KUKA KRL program: TRIGBACK.src

&ACCESS RV
&REL 3
&PARAM TEMPLATE = C:\KRC\Roboter\Template\FunctionVorgabe
&PARAM EDITMASK = *
DEFFCT BOOL TRIGBACK( )

DECL STIFFNESS USERSTIFF

DECL INT md_int[16]
DECL REAL md_real[16]
DECL INT n
DECL INT result

;USERSTIFF=$STIFFNESS
;USERSTIFF.STRATEGY=10
;USERSTIFF.FRAMETYPE=#TOOL
;USERSTIFF.TOOL={X 0.0,Y 0.0,Z 180.0,A 0.0,B 0.0,C 0.0}
;USERSTIFF.CPSTIFFNESS={X 2000,Y 2000,Z 2000,A 200,B 200,C 200}
;USERSTIFF.CPDAMPING={X 0.7,Y 0.7,Z 0.7,A 0.7,B 0.7,C 0.7}
;USERSTIFF.AXISSTIFFNESS={A1 2000,A2 2000,A3 2000,A4 2000,A5 2000,A6 2000,E1 2000}
;USERSTIFF.AXISDAMPING={A1 0.7,A2 0.7,A3 0.7,A4 0.7,A5 0.7,A6 0.7,E1 0.7}
;USERSTIFF.CPMAXDELTA={X 7.0,Y 7.0,Z 7.0,A 2.0,B 2.0,C 2.0}
;USERSTIFF.MAXFORCE={X 70,Y 70,Z 70,A 10,B 10,C 10}
;USERSTIFF.AXISMAXDELTA={A1 10,A2 10,A3 10,A4 10,A5 10,A6 10,E1 10}
;USERSTIFF.AXISMAXDELTATRQ={A1 2,A2 2,A3 2,A4 2,A5 2,A6 2,E1 2}

FOR n=1 TO 16
md_int[n]=0
md_real[n]=0
ENDFOR

md_real[1]=0.05

result=MD_CMD("PAPAS","TRIGBYCONTACT",md_int[],md_real[])

RETURN TRUE
ENDFCT
